PROGRAM Axis2_Motion
VAR
	//power
	MC_Power_Axis2: MC_Power;
	//Move
	m_State_Axis2: INT;
	MC_MoveAbsolute_Axis2: MC_MoveAbsolute;

	//JOG
	j_State_Axis2: INT;
	MC_JOG_Axis2: MC_Jog;

	//Stop
	MC_Stop_Axis2: MC_Stop;
	s_State_Axis2: INT;

	//reset
	r_State_Axis2: INT;
	MC_Reset_Axis2: MC_Reset;

	//setposition
	MC_SetPosition_Axis2: MC_SetPosition;
	sp_State_Axis2: INT;
	SetPosition_delay_Axis2:TON;
	//button interlock
	Axis2_J1: BOOL;//JOG+
	Axis2_J2: BOOL;//JOG-
	Axis2_P: BOOL;//Position moving
	Axis2_S: BOOL;//Stop
	Axis2_SP: BOOL;//set position
	//input protect
	Axis2_PositionProtectionSet:BOOL;
	Axis2_InputPositionOutOfRange:BOOL;	
	//
	es_State_Axis2: INT;
	FTrig_ReachLS2: F_TRIG;
	RTrig_EStop2:R_TRIG;
	btn_ReachLSReset_Axis2: BOOL;
END_VAR

//
//输入保护
//
IF btn_Move_Axis2 THEN
	IF targetPositionAxis2>=Axis2_minPosition AND targetPositionAxis2<=Axis2_maxPosition THEN
		Axis2_InputPositionOutOfRange:=FALSE;
		Error:=FALSE;
		ErrorId:=0;
		ErrorDescription:='';
	ELSE
		Axis2_InputPositionOutOfRange:=TRUE;
		Error:=TRUE;
		ErrorId:=1001;
		ErrorDescription:='Axis2_InputPositionOutOfRange';
		RETURN;
	END_IF
END_IF
IF btn_JogForward_Axis2 THEN
	IF Axis2_CurrentPosition_retain+increaseJogPositionAxis2<=Axis2_maxPosition  THEN
		Axis2_InputPositionOutOfRange:=FALSE;
		Error:=FALSE;
		ErrorId:=0;
		ErrorDescription:='';
	ELSE
		Axis2_InputPositionOutOfRange:=TRUE;
		Error:=TRUE;
		ErrorId:=1002;
		ErrorDescription:='exceed Axis2_maxPosition';
		RETURN;
	END_IF
END_IF 

IF  btn_JogBackward_Axis2 THEN
	IF Axis2_CurrentPosition_retain-increaseJogPositionAxis2>=Axis2_minPosition  THEN
		Axis2_InputPositionOutOfRange:=FALSE;
		Error:=FALSE;
		ErrorId:=0;
		ErrorDescription:='';
	ELSE
		Axis2_InputPositionOutOfRange:=TRUE;
		Error:=TRUE;
		ErrorId:=1003;
		ErrorDescription:='less than Axis2_minPosition';
		RETURN;
	END_IF
END_IF
//
//运行状态指示
//
Axis2.ReadStatus();
IF  Axis2.Status.Moving  THEN
	Axis2_moving:=TRUE;
ELSE
	Axis2_moving:=FALSE;
END_IF;
//
//电机错误指示
//
IF  axis2.NcToPlc.ErrorCode=0 THEN
	Axis2_error     := FALSE;
ELSE
	Axis2_error     := TRUE;
	Error:=TRUE;
	ErrorId:=1002;
	ErrorDescription:='axis2.NcToPlc.ErrorCode=0';
END_IF;
//
//Moving_done_Axis2
//
//
Moving_done_Axis2:=MC_MoveAbsolute_Axis2.Done OR MC_JOG_Axis2.Done;
//
//Positioning move
//
A_MCAxis2();
CASE m_State_Axis2 OF 
	0:
		//检查是否有错误等
		IF  NOT Axis2_error THEN
			m_State_Axis2:=1;
		ELSE
			m_State_Axis2:=-100;
		END_IF
	1:
		//检查电机是否已经上电，如无，则上电
		IF 	NOT MC_Power_Axis2.Status THEN
			MC_Power_Axis2.Enable:=TRUE;
		ELSE
			m_State_Axis2:=2;
		END_IF
	2:
		//定位运行
		MC_MoveAbsolute_Axis2.Position:=targetPositionAxis2;
		MC_MoveAbsolute_Axis2.Velocity:=targetVelocityAxis2;
		IF btn_Move_Axis2 THEN
			MC_MoveAbsolute_Axis2.Execute:=TRUE;
			m_State_Axis2:=3;
		END_IF
	3:
		//是否运动到位
		IF MC_MoveAbsolute_Axis2.Done THEN
			m_State_Axis2:=88;
		END_IF
	88:
		btn_Move_Axis2:=FALSE;
		MC_MoveAbsolute_Axis2.Execute:=FALSE;
		m_State_Axis2:=0;		
	-100:
		btn_Move_Axis2:=FALSE;
		MC_MoveAbsolute_Axis2.Execute:=FALSE;
		Error:=TRUE;
		Axis2_error:=TRUE;
		ErrorId:=1002;
		ErrorDescription:='Axis2 move error';
		
END_CASE
//
//JOG+
//
CASE j_State_Axis2 OF 
	0:
		//检查是否有错误等
		IF  NOT Axis2_error THEN
			j_State_Axis2:=1;
		ELSE
			j_State_Axis2:=-100;
		END_IF
	1:
		//检查电机是否已经上电，如无，则上电
		IF 	NOT MC_Power_Axis2.Status THEN
			MC_Power_Axis2.Enable:=TRUE;
		ELSE
			j_State_Axis2:=2;
		END_IF
	2:
		//JOG运行
		MC_JOG_Axis2.Position:=increaseJogPositionAxis2;
		MC_JOG_Axis2.Velocity:=targetVelocityAxis2;
		IF btn_JogForward_Axis2 AND NOT btn_JogBackward_Axis2 THEN
			MC_JOG_Axis2.JogForward:=TRUE;
			j_State_Axis2:=3;
		END_IF
		IF btn_JogBackward_Axis2 AND NOT btn_JogForward_Axis2 THEN
			MC_JOG_Axis2.JogBackwards:=TRUE;
			j_State_Axis2:=3;
		END_IF
	3:
		//是否运动到位
		IF btn_JogForward_Axis2 THEN
			btn_JogForward_Axis2:=FALSE;
		END_IF 
		IF btn_JogBackward_Axis2 THEN
			btn_JogBackward_Axis2:=FALSE;
		END_IF
		IF MC_JOG_Axis2.Done THEN
			j_State_Axis2:=88;
		END_IF
	88:
		MC_JOG_Axis2.JogForward:=FALSE;
		MC_JOG_Axis2.JogBackwards:=FALSE;
		btn_JogForward_Axis2:=FALSE;
		btn_JogBackward_Axis2:=FALSE;
		j_State_Axis2:=0;	
		
	-100:
		MC_JOG_Axis2.JogForward:=FALSE;
		MC_JOG_Axis2.JogBackwards:=FALSE;
		btn_JogForward_Axis2:=FALSE;
		btn_JogBackward_Axis2:=FALSE;
		Error:=TRUE;
		Axis2_error:=TRUE;
		ErrorId:=1002;
		ErrorDescription:='Axis2 jog error';	
END_CASE
//
//STOP
//
CASE s_State_Axis2 OF 
	0:
		s_State_Axis2:=1;
	1:
		//检查电机是否已经上电，如无，则上电
		IF 	NOT MC_Power_Axis2.Status THEN
			MC_Power_Axis2.Enable:=TRUE;
		ELSE
			s_State_Axis2:=2;
		END_IF
	2:
		//STOP
		IF btn_Stop_Axis2 THEN
			MC_Stop_Axis2.Execute:=TRUE;
			s_State_Axis2:=3;
		END_IF
	3:
		//是否运动到位
		IF MC_Stop_Axis2.Done THEN
			s_State_Axis2:=88;
		END_IF
	88:
		btn_Stop_Axis2:=FALSE;
		MC_Stop_Axis2.Execute:=FALSE;
		s_State_Axis2:=0;	
		//reset status
		btn_Move_Axis2:=FALSE;
		MC_MoveAbsolute_Axis2.Execute:=FALSE;
		btn_JogForward_Axis2:=FALSE;
		btn_JogBackward_Axis2:=FALSE;
		MC_JOG_Axis2.JogForward:=FALSE;
		MC_JOG_Axis2.JogBackwards:=FALSE;
		m_State_Axis2:=0;
		j_State_Axis2:=0;
	-100:
		btn_Stop_Axis2:=FALSE;
		MC_Stop_Axis2.Execute:=FALSE;
		Error:=TRUE;
		Axis2_error:=TRUE;
		ErrorId:=1002;
		ErrorDescription:='Axis2 stop error';
		//reset status
		btn_Move_Axis2:=FALSE;
		MC_MoveAbsolute_Axis2.Execute:=FALSE;
		btn_JogForward_Axis2:=FALSE;
		btn_JogBackward_Axis2:=FALSE;
		MC_JOG_Axis2.JogForward:=FALSE;
		MC_JOG_Axis2.JogBackwards:=FALSE;
		m_State_Axis2:=0;
		j_State_Axis2:=0;
END_CASE
//
//Reset
//
CASE r_State_Axis2 OF 
	0:
		IF btn_Reset_Axis2 OR btn_ReachLSReset_Axis2 THEN
			MC_Reset_Axis2.Execute:=TRUE;
			r_State_Axis2:=1;
		END_IF
	1:
		//是否运动到位
		IF MC_Reset_Axis2.Done THEN
			r_State_Axis2:=88;
		END_IF
	88:
		r_State_Axis2:=0;
		MC_Reset_Axis2.Execute:=FALSE;	
		btn_Reset_Axis2:=FALSE;
		btn_ReachLSReset_Axis2:=FALSE;
		//reset status
		btn_Move_Axis2:=FALSE;
		MC_MoveAbsolute_Axis2.Execute:=FALSE;
		btn_JogForward_Axis2:=FALSE;
		btn_JogBackward_Axis2:=FALSE;
		MC_JOG_Axis2.JogForward:=FALSE;
		MC_JOG_Axis2.JogBackwards:=FALSE;
		m_State_Axis2:=0;
		s_State_Axis2:=0;
		j_State_Axis2:=0;
END_CASE
//
//setposotion
//
SetPosition_delay_Axis2.PT:=T#0.1S;
SetPosition_delay_Axis2();
IF btn_SetPosition_Axis2 THEN
	CASE sp_State_Axis2 OF 
		0:
			IF NOT Axis2_moving THEN
				sp_State_Axis2:=1;
			END_IF
		1:
			MC_SetPosition_Axis2.Position:=PositionSetValue_Axis2;
			MC_SetPosition_Axis2.Execute:=TRUE;
			SetPosition_delay_Axis2.IN:=TRUE;
			sp_State_Axis2:=2;
		2:
			IF MC_SetPosition_Axis2.Done THEN
				sp_State_Axis2:=88;
			END_IF
			IF SetPosition_delay_Axis2.Q THEN//延时结束时，还没有设置位置成功
				sp_State_Axis2:=-100;
			END_IF
		88:
			PositionSetDone_Axis2:=TRUE;
			MC_SetPosition_Axis2.Execute:=FALSE;
			SetPosition_delay_Axis2.IN:=FALSE;
			sp_State_Axis2:=0;
			btn_SetPosition_Axis2:=FALSE;
		-100:
			PositionSetDone_Axis2:=FALSE;
			MC_SetPosition_Axis2.Execute:=FALSE;
			SetPosition_delay_Axis2.IN:=FALSE;
			btn_SetPosition_Axis2:=FALSE;
	END_CASE
END_IF
//
//
//
//急停
IF NOT(E_STOP AND E_STOP_rem AND Plc_EmergencyStop) THEN
	CASE es_State_Axis2 OF
		0:
			es_State_Axis2:=1;
		1:
			E_STOP_led:= FALSE;	//red
			MC_Power_Axis2.Enable:=FALSE;//电机2断电
			btn_Stop_Axis2:=TRUE;//STOP axis1
			A_MCAxis2();
			Error:=TRUE;
			ErrorId:=101;
			ErrorDescription:='E_STOP';
	END_CASE
ELSE
		E_STOP_led:= TRUE;	//green
		//Error:=FALSE;
		//ErrorId:=0;
		//ErrorDescription:='';
END_IF
RTrig_EStop2(CLK:=E_STOP AND E_STOP_rem AND Plc_EmergencyStop);
IF RTrig_EStop2.Q THEN
	E_STOP_led:= TRUE;	//green
	Error:=FALSE;
	ErrorId:=0;
	ErrorDescription:='';
END_IF


(*触发限位开关后，相当于点击了Stop按钮*)
FTrig_ReachLS2(CLK:=foreward_limit_axis2 AND backward_limit_axis2);
IF FTrig_ReachLS2.Q THEN
	btn_Reset_Axis2:=TRUE;
	btn_ReachLSReset_Axis2:=TRUE;
END_IF


//
//屏幕按钮**互锁变量,FALSE时，该按钮灰色不能触发
//
//J1->JOG+
IF  foreward_limit_axis2 AND E_STOP  AND Local_led AND NOT  Axis2_error  AND NOT  Axis2_moving AND
	NOT btn_Move_Axis2 AND NOT  btn_JogBackward_Axis2  THEN
	Axis2_J1     := TRUE;
ELSE
	Axis2_J1     := FALSE;
END_IF;
//J2>JOG-
IF  backward_limit_axis2  AND E_STOP   AND Local_led AND NOT  Axis2_error  AND NOT  Axis2_moving AND 
	 NOT  btn_Move_Axis2 AND NOT btn_JogForward_Axis2 THEN
	Axis2_J2     := TRUE;
ELSE
	Axis2_J2     := FALSE;
END_IF;
//P->PositionMove
IF  E_STOP   AND Local_led AND NOT  Axis2_error  AND NOT  Axis2_moving AND 
	 NOT btn_JogForward_Axis2  AND NOT  btn_JogBackward_Axis2 THEN
	Axis2_P     := TRUE;
ELSE
	Axis2_P     := FALSE;
END_IF;
//SP->SetPosition
IF E_STOP  AND Local_led AND NOT  Axis2_error  AND NOT Axis2_moving  THEN
	Axis2_SP     := TRUE;
ELSE
	Axis2_SP     := FALSE;
END_IF;
//S->Stop
IF E_STOP  AND Local_led AND NOT  Axis2_error THEN
	Axis2_S     := TRUE;
ELSE
	Axis2_S     := FALSE;
END_IF;

ACTION A_MCAxis2:
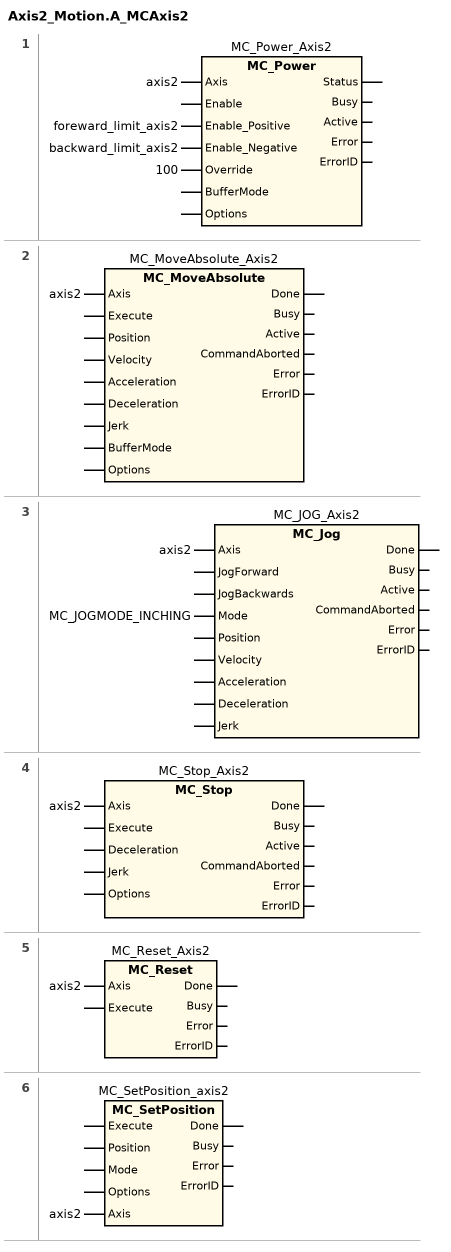
// NETWORK 1
MC_Power_Axis2(
    Axis := axis2,
    Enable_Positive := foreward_limit_axis2,
    Enable_Negative := backward_limit_axis2,
    Override := 100); // MC_Power

// NETWORK 2
MC_MoveAbsolute_Axis2(Axis := axis2); // MC_MoveAbsolute

// NETWORK 3
MC_JOG_Axis2(Axis := axis2, Mode := MC_JOGMODE_INCHING); // MC_Jog

// NETWORK 4
MC_Stop_Axis2(Axis := axis2); // MC_Stop

// NETWORK 5
MC_Reset_Axis2(Axis := axis2); // MC_Reset

// NETWORK 6
MC_SetPosition_axis2(Axis := axis2); // MC_SetPosition
END_ACTION

END_PROGRAM

(* stored: Version 1.1.0.1, ProductVersion 3.1.4024.6
   POU Axis2_Motion: Id {097146e8-d72b-4f21-bc71-dffd24420c23}, SpecialFunc None
   Action A_MCAxis2: Id {b024b50a-846f-42b5-9fd1-a325677feb88} *)
